{attribute 'qualified_only'}
{attribute 'strict'}
TYPE ST110_PnpVerPos_e :
(
    UpEmpty,               // Up position when the Pnp is empty
    DownEmpty,             // Down position when the Pnp is picking the piece
    UpFull,                // Up position when the Pnp has gripped the piece
    DownFullQuick,         // down position with quick speed
    DownFullTorqueControl, // down position with low speed for torque control
    _max
);
END_TYPE

(* stored: Version 1.1.0.1, ProductVersion 3.1.4024.6
   DUT ST110_PnpVerPos_e: Id {ec2150e1-bde0-414a-b93a-aeac75a814a7} *)
